{attribute 'qualified_only'}
{attribute 'strict'}
TYPE E_LiquidType :
(
	WATER := 0,
	HONEY,
	SODA
);
END_TYPE

(* stored: Version 1.1.0.1, ProductVersion 3.1.4024.16
   DUT E_LiquidType: Id {d1b9d34c-4b8c-40ef-8256-8b01ae72d3ed} *)
